PROGRAM MAIN
VAR
	fAmount1 : REAL;
	fAmount2 : REAL;
	fbBank : FB_Bank;
	fbIciciBank : FB_IciciBank;
END_VAR

//fAmount1 := fbBank.fMoney;
fbBank.sBankName := 'sbi';
fbBank.M_Deposit(4000);
fbBank.M_Withdrawal(2000);
//fAmount2 := fbIciciBank.fMoney;
fbIciciBank.sBankName := 'icici';
//fbIciciBank.M_Deposit(4000);
//fbIciciBank.M_Withdrawal(2000);
fbIciciBank.Test();
fbIciciBank.nNum1 := 32;
fbBank();

END_PROGRAM

(* stored: Version 1.1.0.1, ProductVersion 3.1.4024.16
   POU MAIN: Id {01142b65-2ce5-4b19-885c-dce016012905}, SpecialFunc None
   Folder VISUs: Id {c4dd43bf-d2ea-4409-a659-a04952fc54ed} *)
